FUNCTION_BLOCK ABSTRACT FB_Vehicle

VAR
		sOutput : STRING;
END_VAR

METHOD ABSTRACT Speed
VAR_INPUT
END_VAR
END_METHOD

METHOD ABSTRACT VehicleName
VAR_INPUT
END_VAR
END_METHOD

END_FUNCTION_BLOCK

(* stored: Version 1.1.0.1, ProductVersion 3.1.4024.16
   POU FB_Vehicle: Id {4c43a313-ee16-437a-8b82-ef5ed4134457}, SpecialFunc None
   Method Speed: Id {5054b709-307e-4b93-bf1d-f40b9f285e37}
   Method VehicleName: Id {af49db2e-2bc0-4469-99c4-c2942b2aff3f} *)
